Omron CX-Programmer project NuovoProgetto (CX-Programmer 9.61)

# PLC NewPLC1: CJ2M CPU32
I/O table (CPU CJ2M-CPU32): rack 0 slot 11 CJ2M-EIP21

## Global symbols (name address type ; comment)
AnnoNecessario D700 INT  ; 1° Word di lavoro - Anno di produzione
AnnoNecessarioRicetta D300 INT
AutCmdNotturno W20.07 BOOL
AutCmdStop W20.06 BOOL
AutFlagConforme W20.08 BOOL
AutPoupupAcido W21.02 BOOL
AutPoupupBedina D6122 INT
AutPoupupScolaggio W21.00 BOOL
AutPoupupTBedina D6123 INT
AutPrepBedina W20.08 BOOL
AutPupupInvioBotte D1100.04 BOOL
AutRicettaENd W21.01 BOOL
AutStsScolaggioEnd 6.08 BOOL
0.04 BOOL  ; PER VIS DISPLAY
10.00 BOOL  ; SPIA DISPLAY
10.01 BOOL  ; SPIA DISPLAY
10.03 BOOL  ; SPIA DISPLAY
11.00 BOOL  ; mixA
11.01 BOOL  ; in da rete
11.02 BOOL  ; acqua fredda
11.03 BOOL  ; mixB
11.06 BOOL  ; reset prenotazio
15.00 BOOL  ; ELETTROV_GENERALE
15.01 BOOL  ; EV SCOLAGGIO
15.04 BOOL  ; LUCE VERDE
15.05 BOOL  ; LUCE ROSSA
15.06 BOOL  ; elettrov. mix A
15.07 BOOL  ; ELETTROVALVOLA VAPORE
15.08 BOOL  ; EV SCARICO VASCA
15.09 BOOL  ; EV CARICO VASCA
15.10 BOOL  ; MARCIA AV
15.11 BOOL  ; RELE AGITATORE
15.12 BOOL  ; freno botte
15.13 BOOL  ; AUX POMPA
15.14 BOOL  ; AUX ROTAZ. FILTRO
15.15 BOOL  ; MARCIA IN
204.00 BOOL  ; PER_VIS_DISPLAY
207.00 BOOL  ; SPIA DISPLAY
207.01 BOOL  ; SPIA DISPLAY
20.09 BOOL  ; Fp carica
20.10 BOOL  ; Fp salva
20.11 BOOL  ; Fp start
20.12 BOOL  ; Fp pausa
211 CHANNEL  ; out per rete
212 CHANNEL  ; out per rete
213 CHANNEL  ; out per rete
220.00 BOOL  ; out per rete
220.01 BOOL  ; out per rete
220.02 BOOL  ; out per rete
220.03 BOOL  ; out per rete
220.04 BOOL  ; out per rete
220.05 BOOL  ; mixA
220.06 BOOL  ; mixB
28.01 BOOL  ; prenota
28.06 BOOL  ; check prenot acq
28.09 BOOL  ; conferma dati fo
28.10 BOOL  ; conferma dati gl
28.11 BOOL  ; tasto start form
28.12 BOOL  ; tasto stop formi
28.13 BOOL  ; tasto start glut
28.14 BOOL  ; tasto stop gluta
30.07 BOOL  ; SEGN. DISPLAY
38.04 BOOL  ; manuale filtro
38.05 BOOL  ; manuale mix B
38.07 BOOL  ; riciclo in attes
3.08 BOOL  ; Comando valvola vapore (?)
40.00 BOOL  ; attesa prenotazi
40.01 BOOL  ; acqua in macchin
40.02 BOOL  ; formico in uso
40.03 BOOL  ; solforico in uso
40.04 BOOL  ; glutaral in uso
40.05 BOOL  ; ingresso formico
40.06 BOOL  ; ingresso glutara
42 CHANNEL  ; Da DeviceNet: litri attuali erogati
6.14 BOOL  ; carico bagno
7.02 BOOL  ; tasto ACQUA
7.03 BOOL  ; a pg quantità
7.08 BOOL  ; on agitatore
7.09 BOOL  ; scarico bagno
8.10 BOOL  ; led formico
8.11 BOOL  ; led solforico
8.12 BOOL  ; led glutaral
9.00 BOOL  ; scelta formico
9.01 BOOL  ; scelta solforico
9.02 BOOL  ; scelta glutaral
9.15 BOOL  ; annullamento sce
D1210 CHANNEL  ; Setpoint litri in DEC
D1212 CHANNEL  ; Litri attuali in DEC
D1250 CHANNEL  ; Secondi mancanti
D1260 CHANNEL  ; Minuti per HMI
D214 CHANNEL  ; Puntatore step
D216 CHANNEL  ; Puntatore Step+1
D300 CHANNEL  ; Passo attuale
D3000 CHANNEL  ; Memoria H0
D3002 CHANNEL  ; Memoria D502
D3102 CHANNEL  ; Puntatore
D502 CHANNEL  ; Cambio pagina lato HMI
D58 CHANNEL  ; °C di erogazione
D59 CHANNEL  ; dec/lt in botte
D600 CHANNEL  ; Passo precedente
D700 CHANNEL  ; Passo successivo
D800 CHANNEL  ; Clear
D85 CHANNEL  ; set +
D86 CHANNEL  ; set -
D92 CHANNEL  ; numero botte
E21005 CHANNEL  ; Puntatore a passo da salvare
E21006 CHANNEL  ; Puntatore per caricamento passo da DB a lavoro
E22002 CHANNEL  ; Passo meno 1
H0 CHANNEL  ; Cambio pagina PLC
H12.00 BOOL  ; timer rotazione
H12.04 BOOL  ; sblocco di prova
H4.13 BOOL  ; relè carico bagn
H4.14 BOOL  ; relè agitatore
H4.15 BOOL  ; relè scarico bag
H5.11 BOOL  ; scarico esterno
H6.01 BOOL  ; start miscelazio
H6.02 BOOL  ; segn acqua in ri
H6.03 BOOL  ; segn acquaA in b
H6.05 BOOL  ; abbandono erogaz
H6.07 BOOL  ; segnalazione pre
H6.08 BOOL  ; start miscelazio
H6.09 BOOL  ; segn acquaB in b
T0140 BOOL  ; Delay discrepanza pagine
T0150 BOOL  ; Delay simulazione cmd acqua
T0151 BOOL  ; Delay simulazione cmd acido formico
T0152 BOOL  ; Delay reset feedback acido formico
T0153 BOOL  ; Delay simulazione cmd glutaraldeide
T0154 BOOL  ; Delay reset feedback glutaraldeide
T0156 BOOL  ; Simulazione riempimento acqua in corso
W24.02 BOOL  ; Memoria comando acqua
BedinaRunning D1103.00 BOOL  ; Preparazione bedina in corso
BedinaTimeEnd D1103.01 BOOL
BedinaTimeRef D1103.03 BOOL
BedinaTimeRun D1103.02 BOOL
CaricaRIcetta W20.01 BOOL  ; Carica ricetta
CmdAcqua 28.01 BOOL
CmdFormico 28.09 BOOL
CmdGlutaral 28.10 BOOL
CmdPIDon 2.11 BOOL
CmdRotAlt 3.01 BOOL
CmdRotAv 1.04 BOOL
CmdRotInd 1.05 BOOL
CmdRotNotte 3.13 BOOL
CmdRotStop 1.03 BOOL
CmdScolaggioDecrementoAsse 4.09 BOOL
CmdScolaggioNormale 4.08 BOOL
CmdTemperaturaOFF 2.13 BOOL
CmdTemperaturaON 2.12 BOOL
CodiceNecessario D750 DINT
CodiceNecessarioRicetta D350 DINT
ConfermaBarcodeLetto D1101.03 BOOL
ConfermaBedina D1100.00 BOOL
ConfermaControllo D1100.07 BOOL
ConfermaInvioBotte D1100.01 BOOL
ConfermaMancatoScolaggio D2000.09 BOOL
ConfermaRotNotte 3.15 BOOL
DelayRotazione D1000 UINT
FeedbackAcqua H6.03 BOOL
FeedbackFormico 40.05 BOOL
FeedbackGlutaral 40.06 BOOL
FeedbackRichiestaFormico 8.10 BOOL
FeedbackRotAlt H4.06 BOOL
FeedbackRotAv 207.00 BOOL
FeedbackRotInd 207.01 BOOL
FeedbackRotNotte 4.03 BOOL
FlagAbilitaScansioni D1810.04 BOOL
FlagIgnoraScansioniFallite D1810.02 BOOL
FlagNascondiTasti 1810.04 BOOL
FlagNuovaScansione D1810.00 BOOL
FlagPrimaScansione D1802.00 BOOL
FlagRiempimentoAcqua D2000.07 BOOL  ; =1 a fine riempimento acqua
FlagRitentaScansioni D1810.03 BOOL
FlagScansioniFallite D1810.01 BOOL
FlagSolido D1102.03 BOOL  ; Per fermata botte inserimento prodotti solidi
FlagStsEnd D1100.02 BOOL
GlobalGreenFlash D1102.02 BOOL
GlobalGreenLight D1102.01 BOOL
GlobalStsRun D1102.00 BOOL  ; =1 se ricetta AUT in marcia
LetturaBarcodeErrata D1101.01 BOOL
LetturaBarcodeOK D1101.02 BOOL
LetturaCodPro D1150 DINT  ; Codice letto da barcode
LetturaPesoDINT D1154 DINT  ; Peso letto da barcode (in INTERO)
LetturaPesoMem D1156 REAL
LetturaPesoREAL D1160 REAL  ; Peso letto da barcode (in REALE)
LetturaRicetta D1152 DINT
LetturaRicettaTemp D1162 DINT
LitriAcqua D57 WORD
MemCodPro D1802 DINT
MemPeso D1806 REAL
MemRicetta D1804 DINT
MemTimSkip D2000.05 BOOL
MinAltPreNotte D40 INT  ; Minuti prima di attivare alternata notte
NumeroScansioni D1808 INT
OreAltPreNotte D39 INT  ; Ore prima di attivare alternata notte
PaginaAtt D502 INT
PassoPuntatore D3100 CHANNEL  ; Passo
PassoPuntatoreINT D3106 INT
PercentualeREAL D1164 REAL
PesoFormico D82 WORD
PesoGlutaral D83 WORD
PesoNecessario D760 REAL
PesoNecessarioRicetta D360 REAL
PopupMancatoScolaggio D2000.08 BOOL  ; =1 se viene attivato un riempimento acqua  e FlagRiempimentoAcqua è già TRUE
PopupRotNotte D2000.04 BOOL
ProdottoErratoIgnora D1101.06 BOOL
ProdottoErratoPopup D1101.05 BOOL
ProdottoErratoRiprova 1101.07 BOOL
PupConfermaInvioBotte D1100.03 BOOL
REAL1000 D1166 REAL
RicAaSca D8000 WORD  ; 1° Word di lavoro - Anno di produzione
RicAzione D8006 WORD  ; Codice azione
RicBotte D8003 WORD  ; Bottale (1-10) di destinazione
RicCheck D8074 WORD  ; Tipo controllo: 1=PH 2=Colore 3=Penetrazione
RicCodPro D8050 DWORD  ; Codice prodotto
RicDescr D8007 STRING[40]  ; Descrizione azione
RicGradi D8064 WORD  ; Temperatura acqua
RicLoaded D8092.00 BOOL  ; 0=nuova 1=ricetta importata
RicMax D8080 REAL  ; Valore massimo per controllo
RicMin D8076 REAL  ; Valore minimo per controllo
RicMinuti D8066 WORD  ; Minuti di rotazione
RicNumSca D8001 DWORD  ; Progressivo ricetta
RicPause W20.04 BOOL  ; Pausa ricetta
RicPeso D8060 REAL  ; Peso prodotto in Kg
RicRata D8054 WORD  ; 1=Raggruppamento prodotti
RicRigNum D8004 WORD  ; Numero progressivo riga
RicRigSot D8005 WORD  ; Numero progressivo sottoriga
RicRilevato D8084 REAL  ; Valore rilevato al controllo
RicRotaz D8068 WORD  ; Tipo di rotazione
RicScola D8070 WORD  ; Tipo di scolatura
RicSpeed D8072 WORD  ; Velocità (da 2 a 8)
RicStart W20.03 BOOL  ; Start ricetta
RicStato D8088 WORD  ; Stato riga
RicStatus D510 WORD
RicStsRun W20.05 BOOL  ; RicStsRun
RicTipPro D8056 WORD  ; L/76=Liquido S/83=Solido
RicUser D8090 WORD  ; ID Utente che convalida la riga
RicValvola D8058 WORD  ; Valvola associata al prodotto
RicettaNecessaria D701 DINT  ; Progressivo ricetta
RicettaNecessariaRicetta D301 DINT
RichiestaConfermaBedina D1101.04 BOOL
RichiestaFormico 9.00 BOOL
RichiestaGlutar 28.08 BOOL
RichiestaLetturaBarcode D1101.00 BOOL
SalvaRicetta W20.00 BOOL  ; Salva ricetta
SceltaFormico 28.07 BOOL
SceltaGlutar 9.02 BOOL
SkipPasso W20.02 BOOL  ; Salta al passo successivo
StatoMacchina D4000 INT
StatoScansione D1800 INT
StsScolaggioDecrementoAsse 5.01 BOOL
StsScolaggioNormale 5.00 BOOL
TempReal D1008 REAL
TemperaturaAcqua D56 CHANNEL
TemperaturaAcquaPerBCD D3200 CHANNEL
TemperaturaMacchina D23 CHANNEL
TimerAcqua1 T0080 TIMER
TimerAcqua2 T0081 TIMER
TimerAcqua3 T0082 TIMER
TimerAcqua4 T0083 TIMER
TimerFormico1 T0070 TIMER
TimerFormico2 T0071 TIMER
TimerFormico3 T0072 TIMER
TimerFormico4 T0073 TIMER
TimerFormico5 T0074 TIMER
TimerFormico6 T0075 TIMER
TimerGlutar1 T0084 TIMER
TimerGlutar2 T0085 TIMER
TimerGlutar3 T0086 TIMER
TimerGlutar4 T0087 TIMER
TimerGlutar5 T0088 TIMER
TimerGlutar6 T0089 TIMER
TimerPIDoff T0100 TIMER
TimerPIDon T0099 TIMER
TimerRotazione T0093 TIMER
TimerRotazione3 T0094 TIMER
TimerRotazione4 T0095 TIMER
TimerRotazione6 T0096 TIMER
TimerRotazione7 T0097 TIMER
TimerRotazione8 T0098 TIMER
TimerSaltaPasso T0102 TIMER  ; 1s minimo per salto passo
TimerScolaggioNormale T0105 TIMER
TimerScolaggioON T0101 TIMER
TimxBedinaDelay D1206 INT
TimxNumeroOre D1200 INT
TimxRicMinuti D1202 INT
TimxTempDelay D1201 INT
Tolleranza D1140 REAL
TolleranzaInf D1144 REAL
TolleranzaSup D1142 REAL
VaiAInvioInBotte D1100.06 BOOL
VelocBotte D1004 WORD
VisibilitàIndietroMan D2000.06 BOOL  ; Visualizza o meno la freccia indietro verso manuale in HMI
acqua_litriErogati D1212 INT
acqua_setpointRicetta D1210 INT
annullaRicetta D1810.11 BOOL
barrieraAperta W24.08 BOOL
barrieraChiusa W24.09 BOOL
barrieraDigIn 14.03 BOOL
cmdScolaggioBotte W24.05 BOOL  ; Comando per scolaggio da procedura solo botte
confermaVaiABedina D1810.08 BOOL
delayAlternataOn W20.14 BOOL
delayPopupControllo T0106 TIMER
flagFineScolaggio D1810.07 BOOL
flagPrimoRiempimento D1810.14 BOOL  ; =1 dopo il primo riempimento d'acqua. torna a 0 dopo uno scolaggio
inserimentoProdottiRunning D1180.09 BOOL
instCreaData creaData
invioConRisciacquoON H4.15 BOOL
invioSenzaRisciacquoON H5.08 BOOL
luceProdotti D100.00 BOOL
memCmdFormico W24.00 BOOL  ; Memoria cmd formico
memCmdGlutaraldeide W24.01 BOOL  ; Memoria cmd glutaraldeide
minutiRimanentiAlternata D31 CHANNEL
offsetRiga1 D1830 INT
offsetRiga2 D1831 INT
offsetRiga3 D1832 INT
offsetRiga4 D1833 INT
offsetRiga5 D1834 INT
offsetRiga6 D1835 INT
popupConfScola W24.07 BOOL
popupPresOpScola W24.06 BOOL
presenzaOpAcido D1810.06 BOOL  ; Conferma presenza operatore per invio acido/glutaral.
rRicStsRun H50.00 BOOL
scrollDown D1810.10 BOOL
scrollUp D1810.09 BOOL
secondiRimanentiAlternata D30 CHANNEL
stopDaBarriera 6.03 BOOL
tempCondStep1 W20.12 BOOL
temperaturaAcquaErogata 43 WORD
temperaturaBotte 2005 WORD
tempoChiamataOperatore D1820 INT
tempoPasso D1836 INT
tempoPassoMem D1837 INT
timerAlternata T0190 TIMER
timerScrollDown T0108 TIMER
timerScrollUp T0107 TIMER
visibPopupPulsanti D1103.04 BOOL  ; Visibilità pulsanti di conferma su pagina automatico
visualizzaKgAcido W24.03 BOOL
visualizzaKgGlutaral W24.04 BOOL

## Program NuovoProgramma1 (cyclic task 0)
Local symbols
BARRIERA_SIC 14.03 BOOL
EMERGENZA_ARIA 14.00 BOOL
LIVELLO_VASCA 14.04 BOOL
PROX_POS 14.01 BOOL
TERMICI 14.02 BOOL

### Section Sezione1

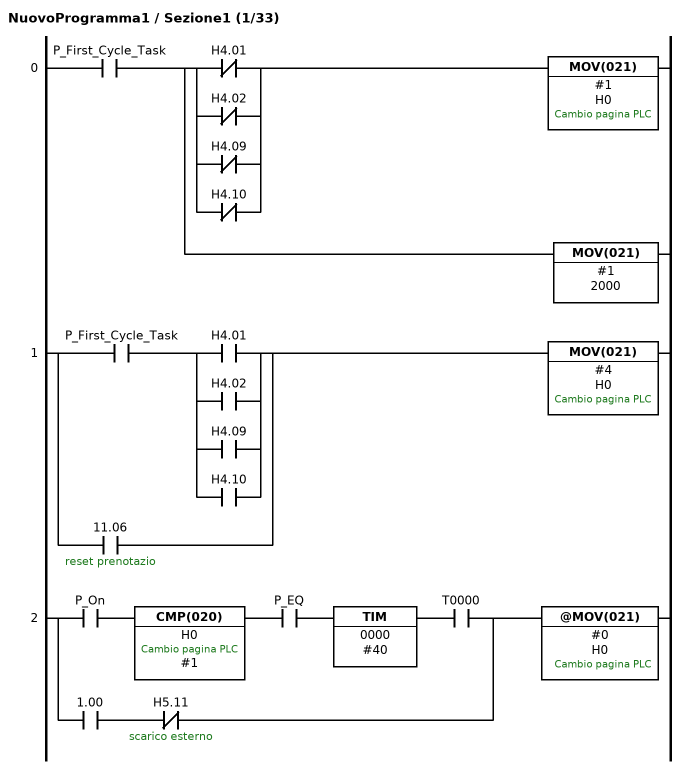
; rung 0
LD P_First_Cycle_Task
OUT TR0
LDNOT H4.01
ORNOT H4.02
ORNOT H4.09
ORNOT H4.10
ANDLD
MOV(021) #1 H0  ; Cambio pagina PLC
LD TR0
MOV(021) #1 2000
; rung 1
LD P_First_Cycle_Task
LD H4.01
OR H4.02
OR H4.09
OR H4.10
ANDLD
OR 11.06  ; reset prenotazio
MOV(021) #4 H0  ; Cambio pagina PLC
; rung 2
LD P_On
CMP(020) H0 #1  ; Cambio pagina PLC
AND P_EQ
TIM 0000 #40
AND T0000
LD 1.00
ANDNOT H5.11  ; scarico esterno
ORLD
@MOV(021) #0 H0  ; Cambio pagina PLC

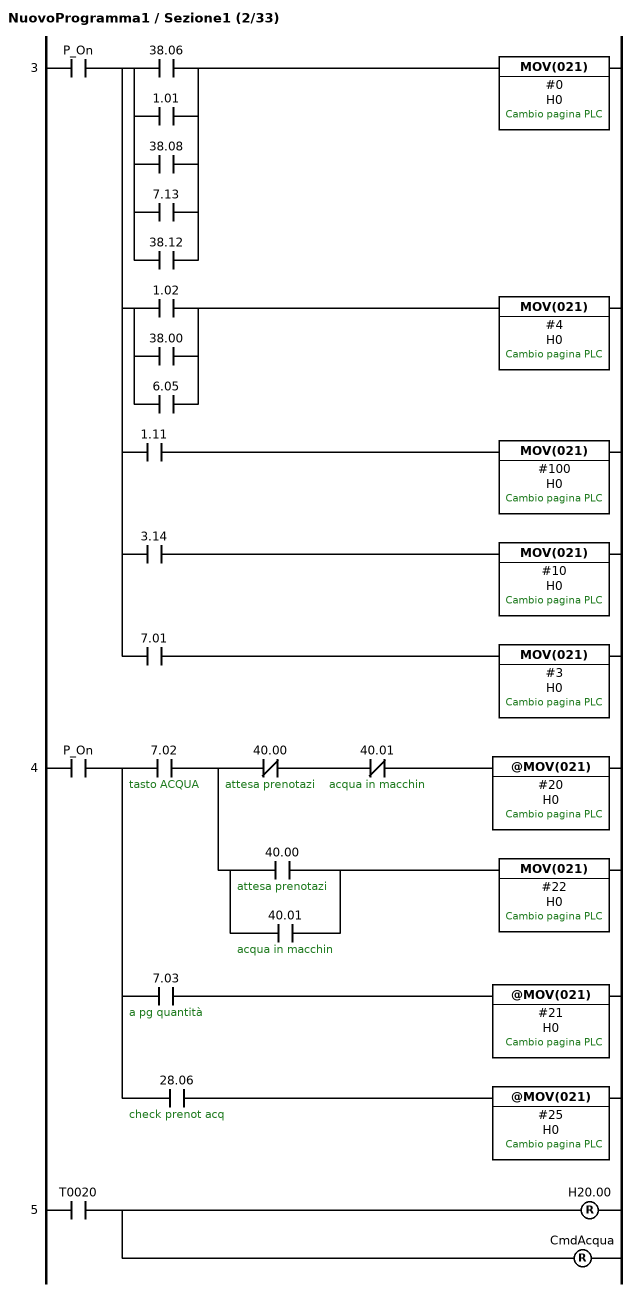
; rung 3
LD P_On
OUT TR0
LD 38.06
OR 1.01
OR 38.08
OR 7.13
OR 38.12
ANDLD
MOV(021) #0 H0  ; Cambio pagina PLC
LD TR0
LD 1.02
OR 38.00
OR 6.05
ANDLD
MOV(021) #4 H0  ; Cambio pagina PLC
LD TR0
AND 1.11
MOV(021) #100 H0  ; Cambio pagina PLC
LD TR0
AND 3.14
MOV(021) #10 H0  ; Cambio pagina PLC
LD TR0
AND 7.01
MOV(021) #3 H0  ; Cambio pagina PLC
; rung 4
LD P_On
OUT TR0
AND 7.02  ; tasto ACQUA
OUT TR1
ANDNOT 40.00  ; attesa prenotazi
ANDNOT 40.01  ; acqua in macchin
@MOV(021) #20 H0  ; Cambio pagina PLC
LD TR1
LD 40.00  ; attesa prenotazi
OR 40.01  ; acqua in macchin
ANDLD
MOV(021) #22 H0  ; Cambio pagina PLC
LD TR0
AND 7.03  ; a pg quantità
@MOV(021) #21 H0  ; Cambio pagina PLC
LD TR0
AND 28.06  ; check prenot acq
@MOV(021) #25 H0  ; Cambio pagina PLC
; rung 5
LD T0020
RSET H20.00
RSET CmdAcqua

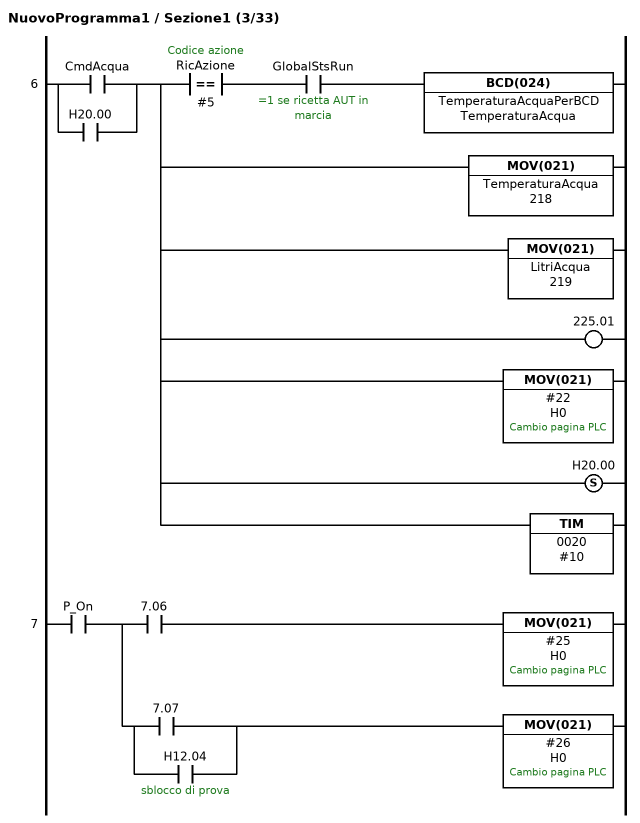
; rung 6
LD CmdAcqua
OR H20.00
OUT TR0
AND=(300) RicAzione #5  ; Codice azione
AND GlobalStsRun  ; =1 se ricetta AUT in marcia
BCD(024) TemperaturaAcquaPerBCD TemperaturaAcqua
LD TR0
MOV(021) TemperaturaAcqua 218
MOV(021) LitriAcqua 219
OUT 225.01
MOV(021) #22 H0  ; Cambio pagina PLC
SET H20.00
TIM 0020 #10
; rung 7
LD P_On
OUT TR0
AND 7.06
MOV(021) #25 H0  ; Cambio pagina PLC
LD TR0
LD 7.07
OR H12.04  ; sblocco di prova
ANDLD
MOV(021) #26 H0  ; Cambio pagina PLC

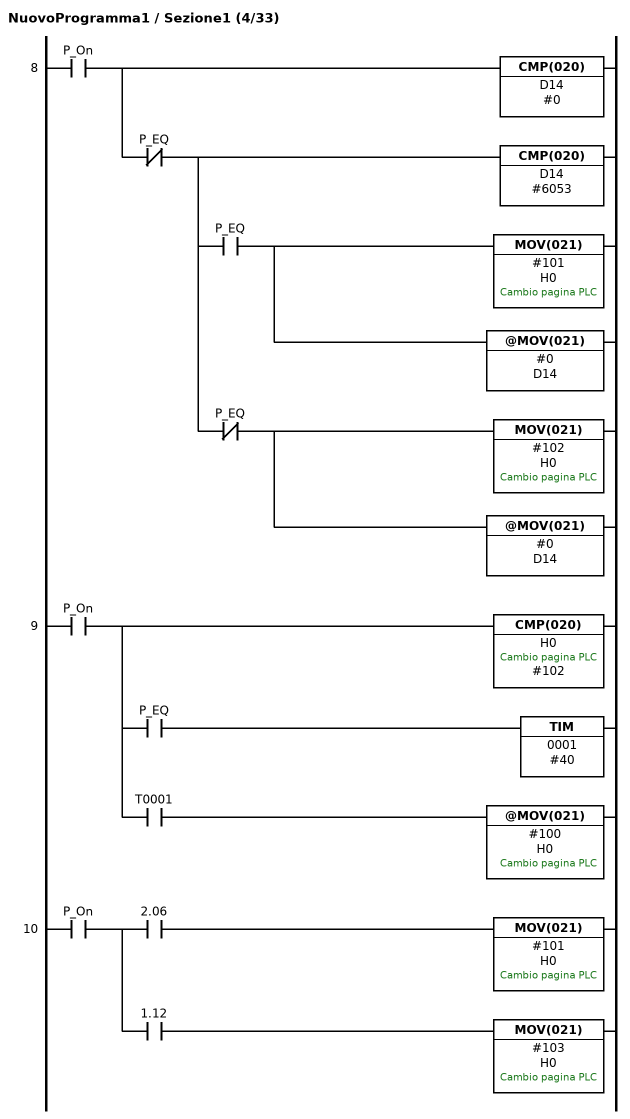
; rung 8
LD P_On
CMP(020) D14 #0
ANDNOT P_EQ
OUT TR0
CMP(020) D14 #6053
AND P_EQ
MOV(021) #101 H0  ; Cambio pagina PLC
@MOV(021) #0 D14
LD TR0
ANDNOT P_EQ
MOV(021) #102 H0  ; Cambio pagina PLC
@MOV(021) #0 D14
; rung 9
LD P_On
OUT TR0
CMP(020) H0 #102  ; Cambio pagina PLC
AND P_EQ
TIM 0001 #40
LD TR0
AND T0001
@MOV(021) #100 H0  ; Cambio pagina PLC
; rung 10
LD P_On
OUT TR0
AND 2.06
MOV(021) #101 H0  ; Cambio pagina PLC
LD TR0
AND 1.12
MOV(021) #103 H0  ; Cambio pagina PLC

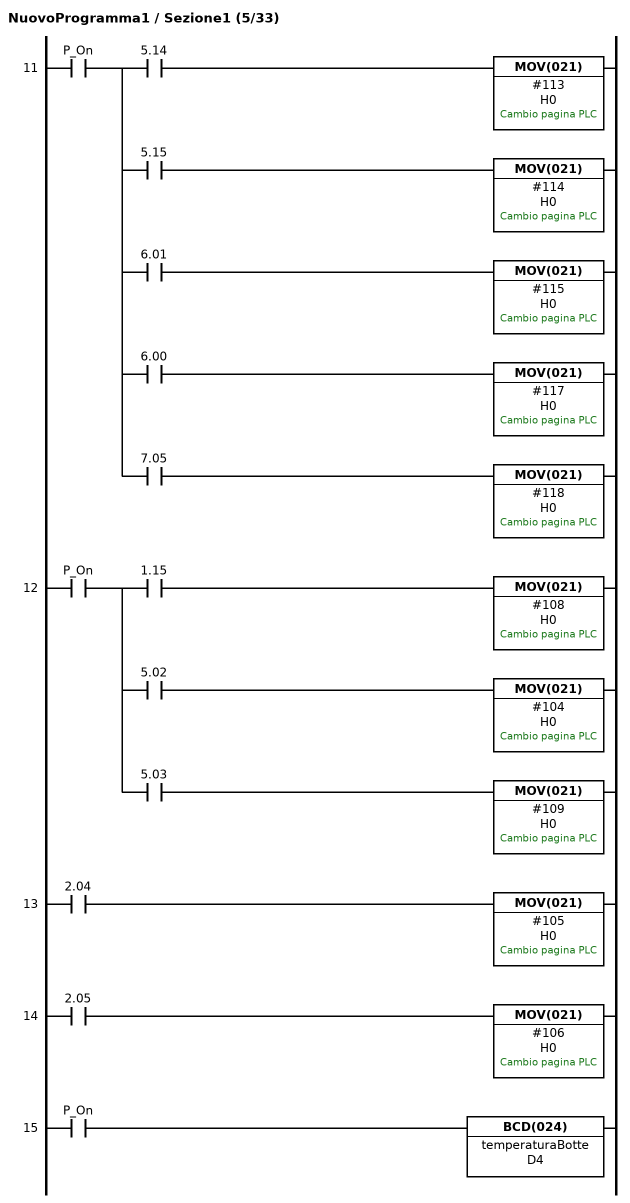
; rung 11
LD P_On
OUT TR0
AND 5.14
MOV(021) #113 H0  ; Cambio pagina PLC
LD TR0
AND 5.15
MOV(021) #114 H0  ; Cambio pagina PLC
LD TR0
AND 6.01
MOV(021) #115 H0  ; Cambio pagina PLC
LD TR0
AND 6.00
MOV(021) #117 H0  ; Cambio pagina PLC
LD TR0
AND 7.05
MOV(021) #118 H0  ; Cambio pagina PLC
; rung 12
LD P_On
OUT TR0
AND 1.15
MOV(021) #108 H0  ; Cambio pagina PLC
LD TR0
AND 5.02
MOV(021) #104 H0  ; Cambio pagina PLC
LD TR0
AND 5.03
MOV(021) #109 H0  ; Cambio pagina PLC
; rung 13
LD 2.04
MOV(021) #105 H0  ; Cambio pagina PLC
; rung 14
LD 2.05
MOV(021) #106 H0  ; Cambio pagina PLC
; rung 15
LD P_On
BCD(024) temperaturaBotte D4

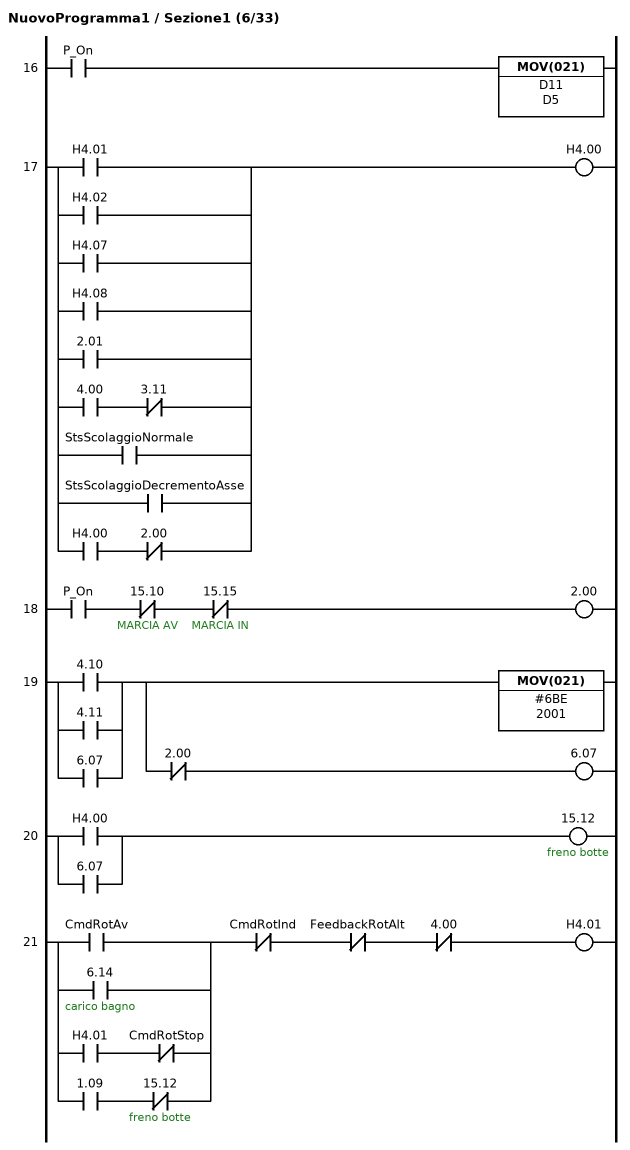
; rung 16
LD P_On
MOV(021) D11 D5
; rung 17
LD H4.01
OR H4.02
OR H4.07
OR H4.08
OR 2.01
LD 4.00
ANDNOT 3.11
ORLD
OR StsScolaggioNormale
OR StsScolaggioDecrementoAsse
LD H4.00
ANDNOT 2.00
ORLD
OUT H4.00
; rung 18
LD P_On
ANDNOT 15.10  ; MARCIA AV
ANDNOT 15.15  ; MARCIA IN
OUT 2.00
; rung 19
LD 4.10
OR 4.11
OR 6.07
MOV(021) #6BE 2001
ANDNOT 2.00
OUT 6.07
; rung 20
LD H4.00
OR 6.07
OUT 15.12  ; freno botte
; rung 21
LD CmdRotAv
OR 6.14  ; carico bagno
LD H4.01
ANDNOT CmdRotStop
ORLD
LD 1.09
ANDNOT 15.12  ; freno botte
ORLD
ANDNOT CmdRotInd
ANDNOT FeedbackRotAlt
ANDNOT 4.00
OUT H4.01

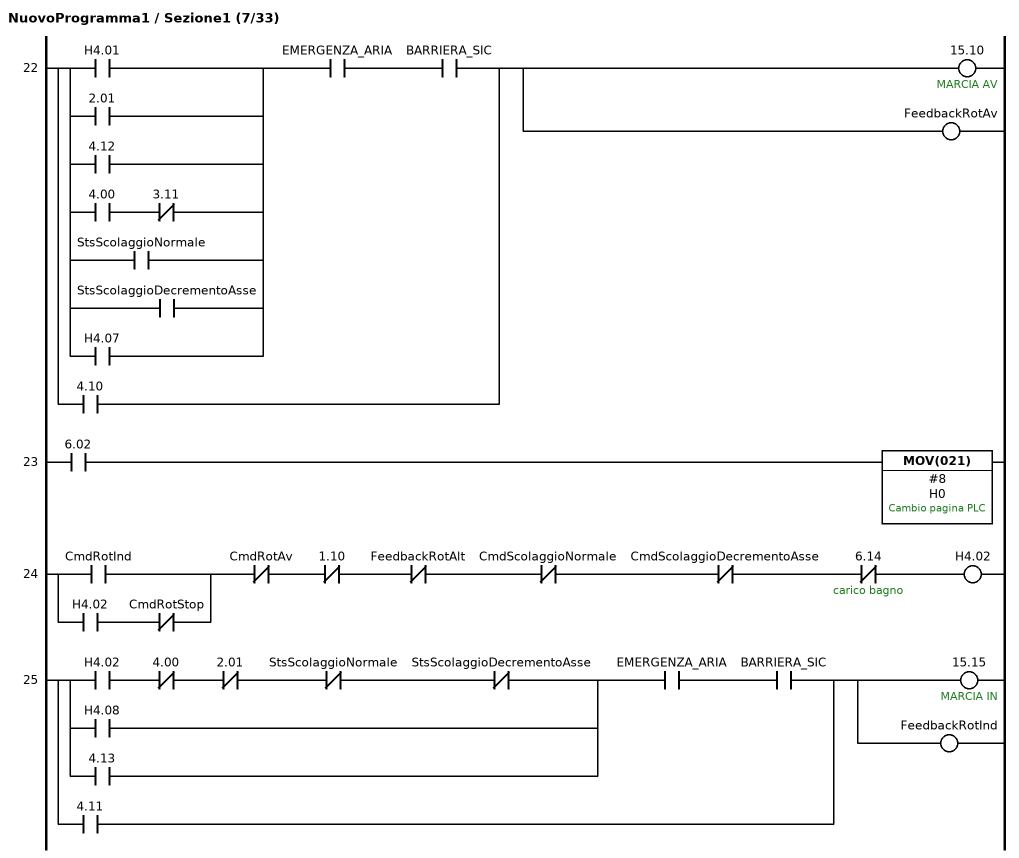
; rung 22
LD H4.01
OR 2.01
OR 4.12
LD 4.00
ANDNOT 3.11
ORLD
OR StsScolaggioNormale
OR StsScolaggioDecrementoAsse
OR H4.07
AND EMERGENZA_ARIA
AND BARRIERA_SIC
OR 4.10
OUT 15.10  ; MARCIA AV
OUT FeedbackRotAv
; rung 23
LD 6.02
MOV(021) #8 H0  ; Cambio pagina PLC
; rung 24
LD CmdRotInd
LD H4.02
ANDNOT CmdRotStop
ORLD
ANDNOT CmdRotAv
ANDNOT 1.10
ANDNOT FeedbackRotAlt
ANDNOT CmdScolaggioNormale
ANDNOT CmdScolaggioDecrementoAsse
ANDNOT 6.14  ; carico bagno
OUT H4.02
; rung 25
LD H4.02
ANDNOT 4.00
ANDNOT 2.01
ANDNOT StsScolaggioNormale
ANDNOT StsScolaggioDecrementoAsse
OR H4.08
OR 4.13
AND EMERGENZA_ARIA
AND BARRIERA_SIC
OR 4.11
OUT 15.15  ; MARCIA IN
OUT FeedbackRotInd

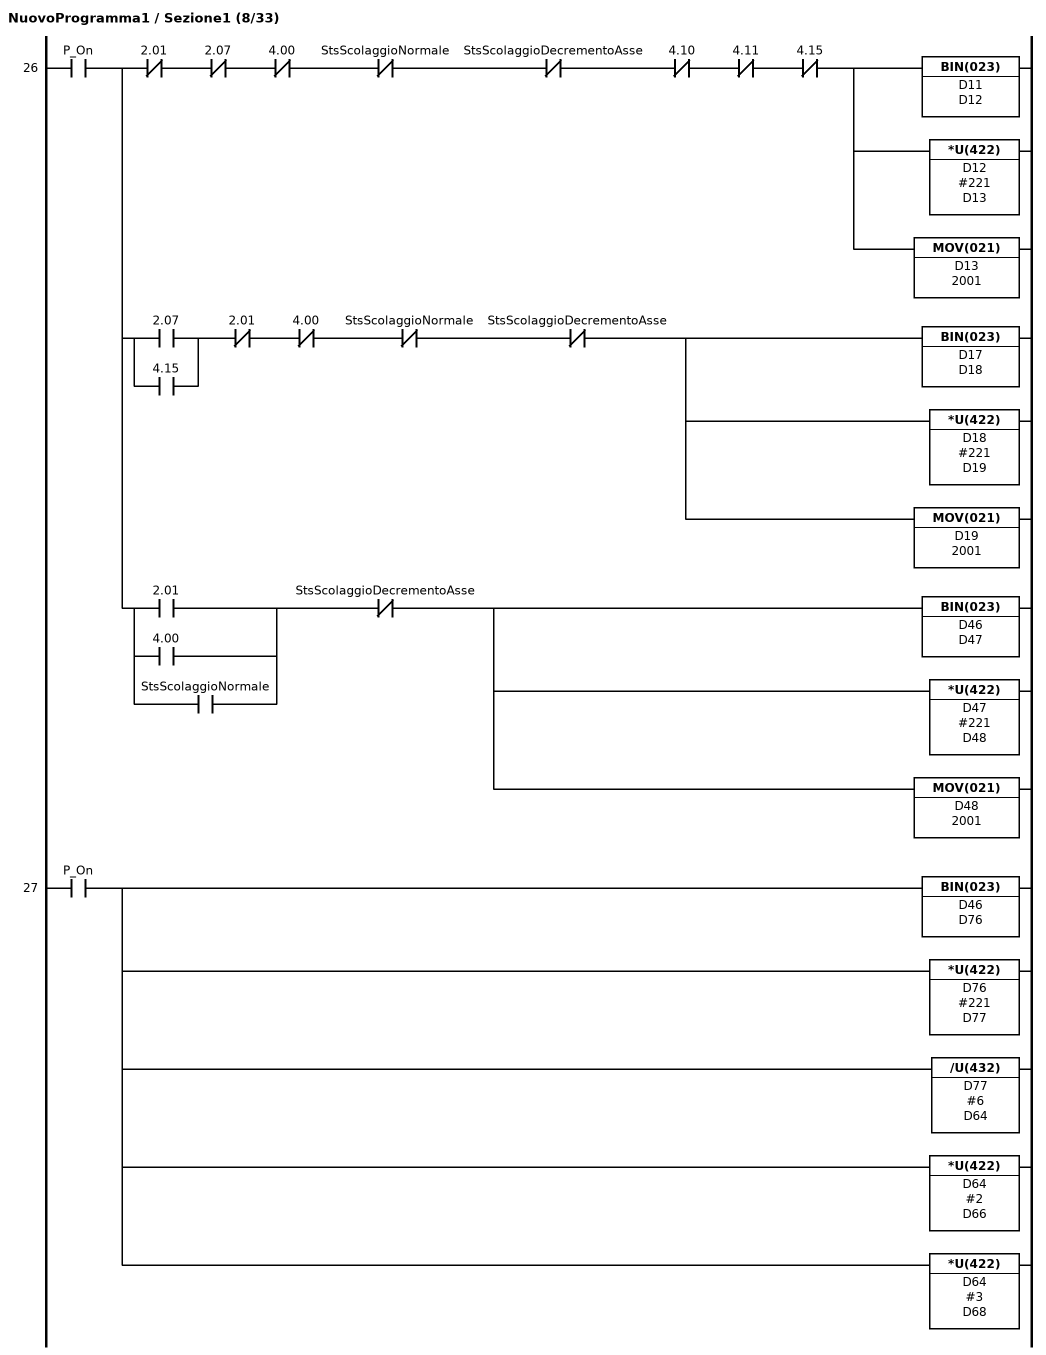
; rung 26
LD P_On
OUT TR0
ANDNOT 2.01
ANDNOT 2.07
ANDNOT 4.00
ANDNOT StsScolaggioNormale
ANDNOT StsScolaggioDecrementoAsse
ANDNOT 4.10
ANDNOT 4.11
ANDNOT 4.15
BIN(023) D11 D12
*U(422) D12 #221 D13
MOV(021) D13 2001
LD TR0
LD 2.07
OR 4.15
ANDLD
ANDNOT 2.01
ANDNOT 4.00
ANDNOT StsScolaggioNormale
ANDNOT StsScolaggioDecrementoAsse
BIN(023) D17 D18
*U(422) D18 #221 D19
MOV(021) D19 2001
LD TR0
LD 2.01
OR 4.00
OR StsScolaggioNormale
ANDLD
ANDNOT StsScolaggioDecrementoAsse
BIN(023) D46 D47
*U(422) D47 #221 D48
MOV(021) D48 2001
; rung 27
LD P_On
BIN(023) D46 D76
*U(422) D76 #221 D77
/U(432) D77 #6 D64
*U(422) D64 #2 D66
*U(422) D64 #3 D68

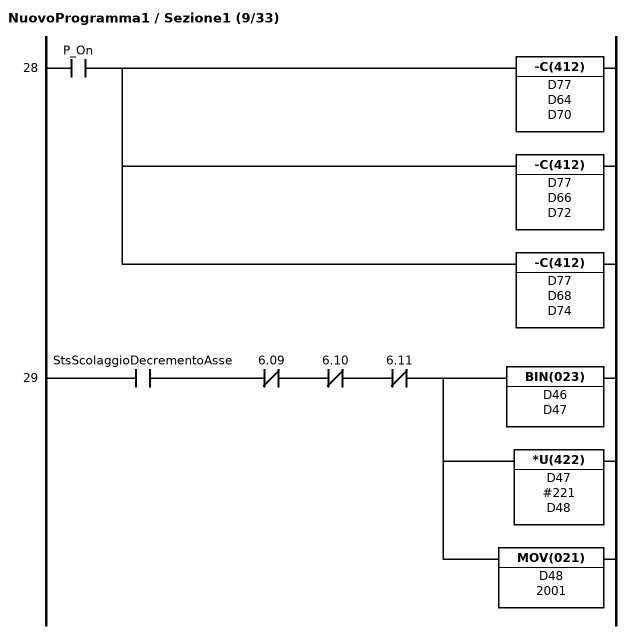
; rung 28
LD P_On
-C(412) D77 D64 D70
-C(412) D77 D66 D72
-C(412) D77 D68 D74
; rung 29
LD StsScolaggioDecrementoAsse
ANDNOT 6.09
ANDNOT 6.10
ANDNOT 6.11
BIN(023) D46 D47
*U(422) D47 #221 D48
MOV(021) D48 2001

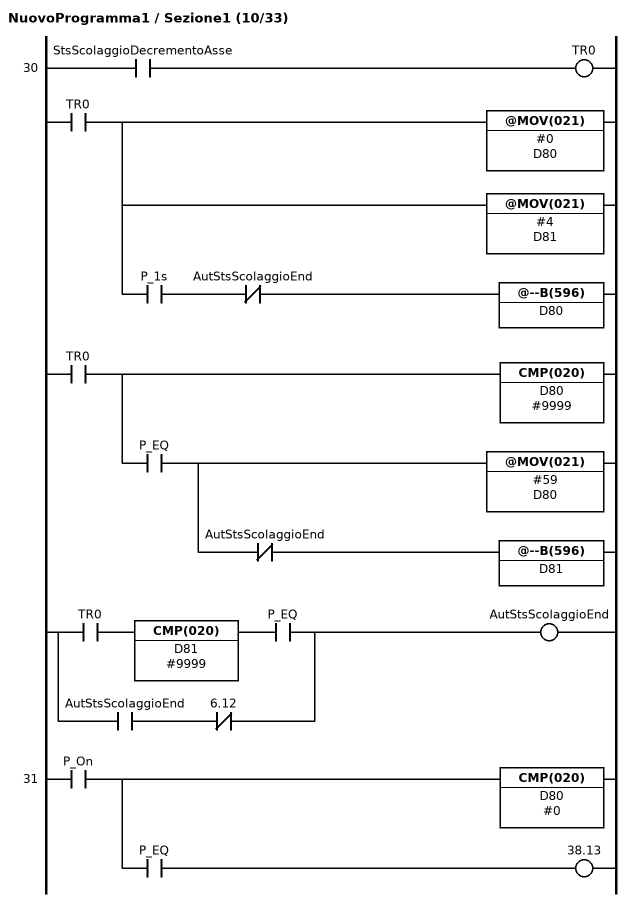
; rung 30
LD StsScolaggioDecrementoAsse
OUT TR0
@MOV(021) #0 D80
@MOV(021) #4 D81
AND P_1s
ANDNOT AutStsScolaggioEnd
@--B(596) D80
LD TR0
CMP(020) D80 #9999
AND P_EQ
@MOV(021) #59 D80
ANDNOT AutStsScolaggioEnd
@--B(596) D81
LD TR0
CMP(020) D81 #9999
AND P_EQ
LD AutStsScolaggioEnd
ANDNOT 6.12
ORLD
OUT AutStsScolaggioEnd
; rung 31
LD P_On
CMP(020) D80 #0
AND P_EQ
OUT 38.13

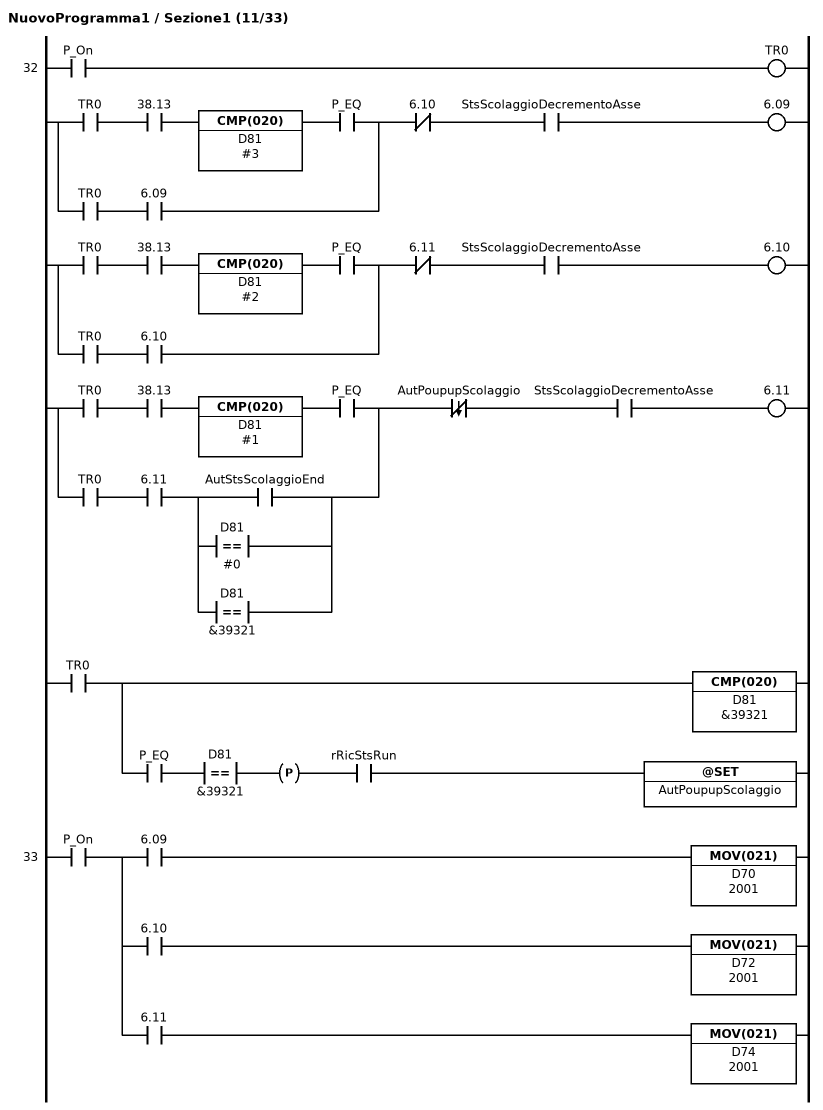
; rung 32
LD P_On
OUT TR0
AND 38.13
CMP(020) D81 #3
AND P_EQ
LD TR0
AND 6.09
ORLD
ANDNOT 6.10
AND StsScolaggioDecrementoAsse
OUT 6.09
LD TR0
AND 38.13
CMP(020) D81 #2
AND P_EQ
LD TR0
AND 6.10
ORLD
ANDNOT 6.11
AND StsScolaggioDecrementoAsse
OUT 6.10
LD TR0
AND 38.13
CMP(020) D81 #1
AND P_EQ
LD TR0
AND 6.11
LD AutStsScolaggioEnd
OR=(300) D81 #0
OR=(300) D81 &39321
ANDLD
ORLD
%ANDNOT AutPoupupScolaggio
AND StsScolaggioDecrementoAsse
OUT 6.11
LD TR0
CMP(020) D81 &39321
AND P_EQ
AND=(300) D81 &39321
UP(521)
AND rRicStsRun
@SET AutPoupupScolaggio
; rung 33
LD P_On
OUT TR0
AND 6.09
MOV(021) D70 2001
LD TR0
AND 6.10
MOV(021) D72 2001
LD TR0
AND 6.11
MOV(021) D74 2001

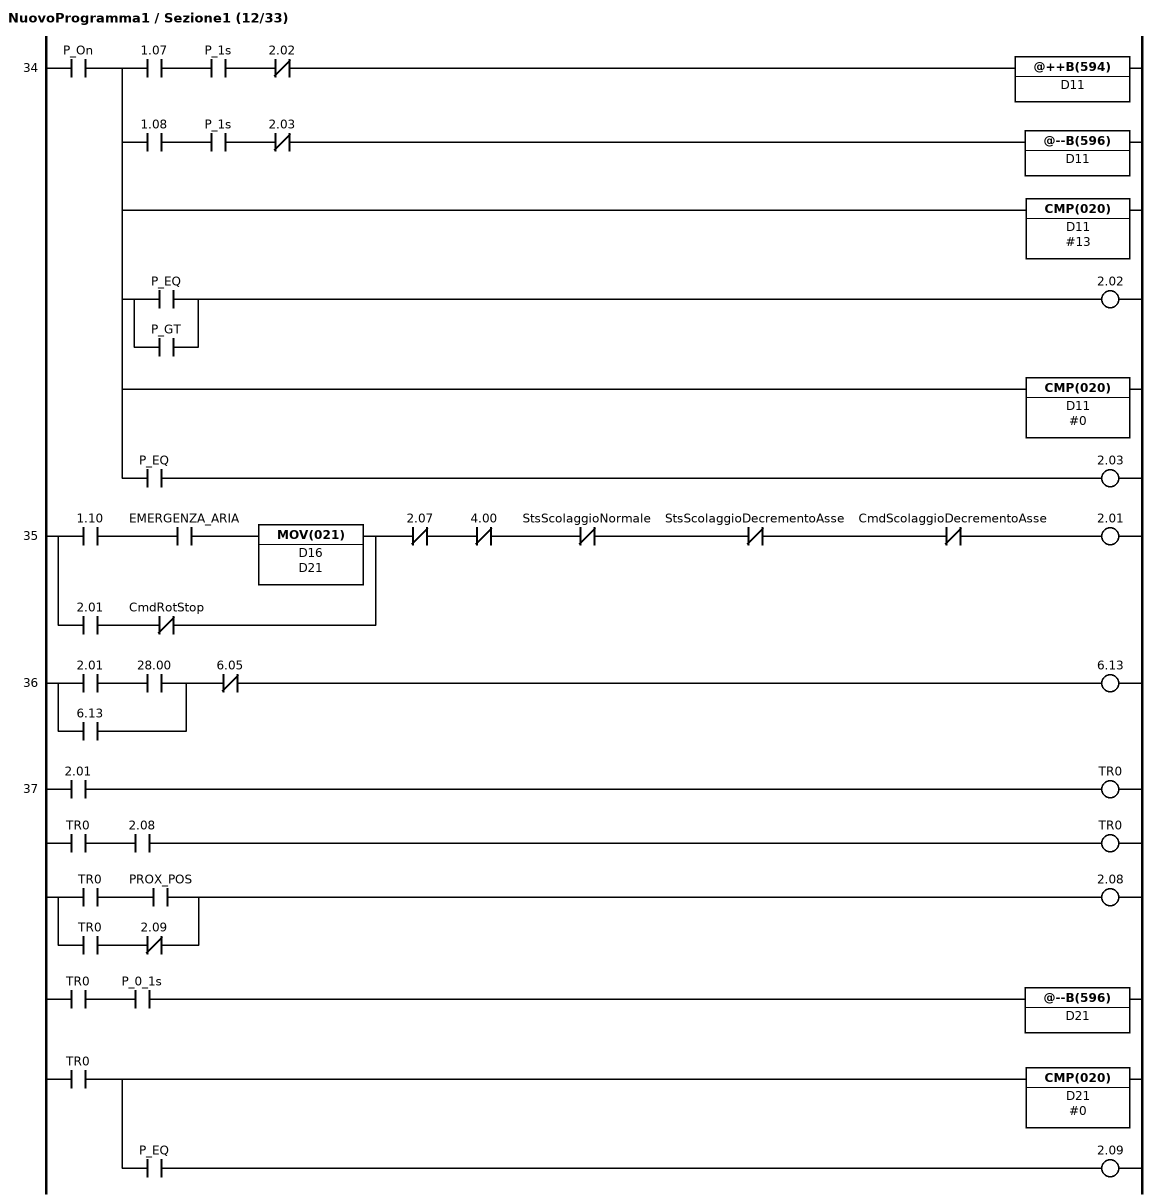
; rung 34
LD P_On
OUT TR0
AND 1.07
AND P_1s
ANDNOT 2.02
@++B(594) D11
LD TR0
AND 1.08
AND P_1s
ANDNOT 2.03
@--B(596) D11
LD TR0
CMP(020) D11 #13
LD P_EQ
OR P_GT
ANDLD
OUT 2.02
LD TR0
CMP(020) D11 #0
AND P_EQ
OUT 2.03
; rung 35
LD 1.10
AND EMERGENZA_ARIA
MOV(021) D16 D21
LD 2.01
ANDNOT CmdRotStop
ORLD
ANDNOT 2.07
ANDNOT 4.00
ANDNOT StsScolaggioNormale
ANDNOT StsScolaggioDecrementoAsse
ANDNOT CmdScolaggioDecrementoAsse
OUT 2.01
; rung 36
LD 2.01
AND 28.00
OR 6.13
ANDNOT 6.05
OUT 6.13
; rung 37
LD 2.01
OUT TR0
AND PROX_POS
LD TR0
AND 2.08
OUT TR0
ANDNOT 2.09
ORLD
OUT 2.08
LD TR0
AND P_0_1s
@--B(596) D21
LD TR0
CMP(020) D21 #0
AND P_EQ
OUT 2.09

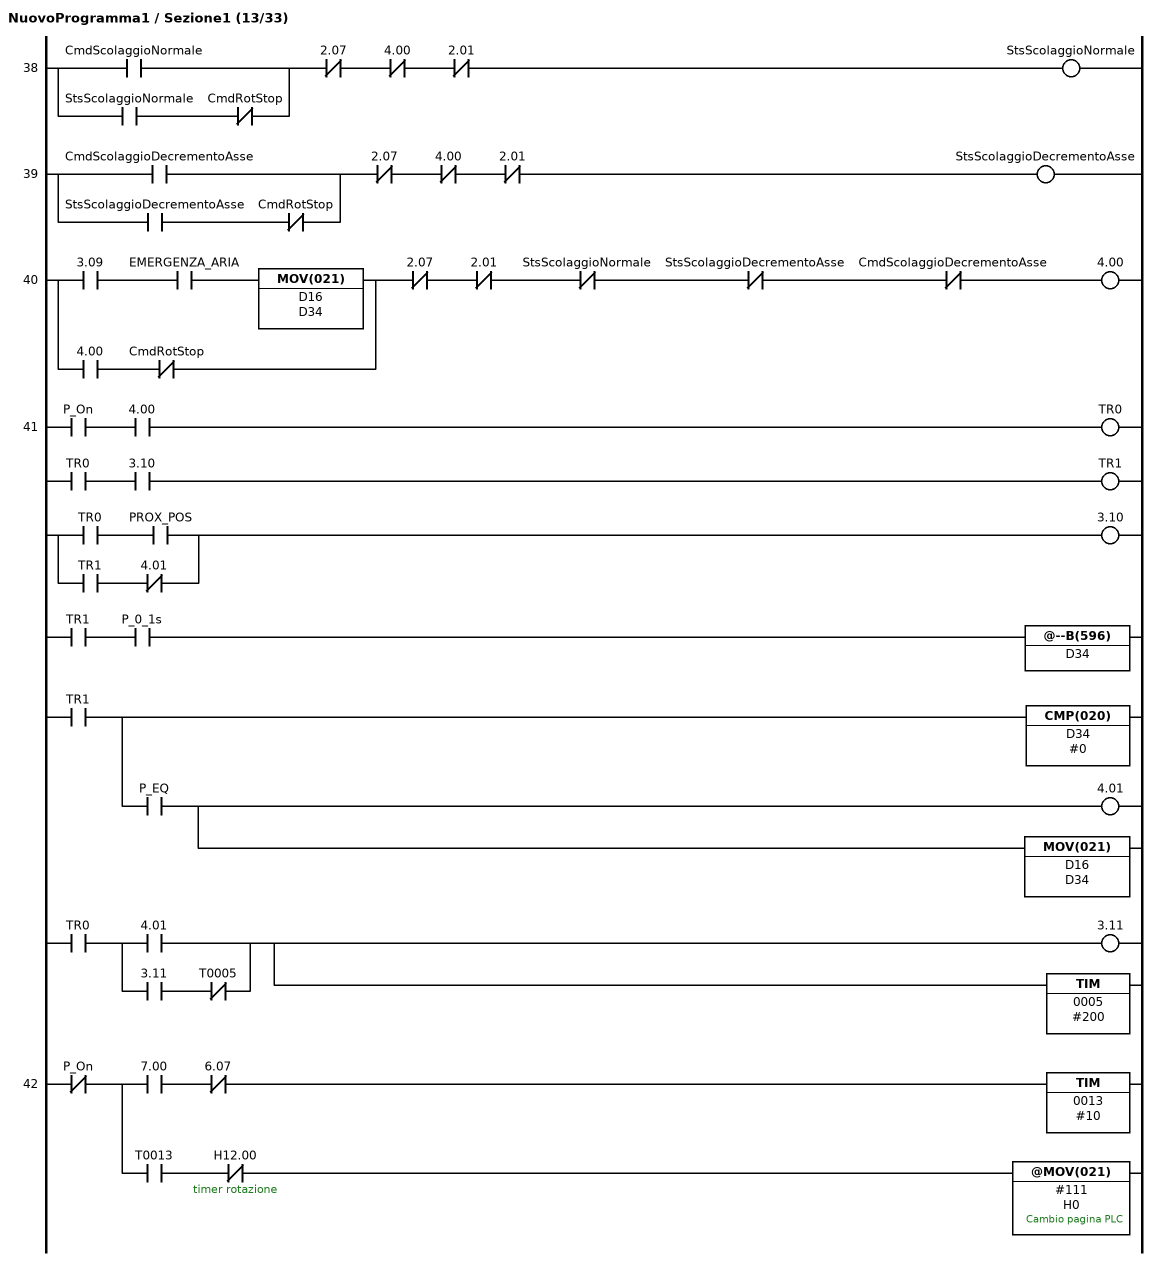
; rung 38
LD CmdScolaggioNormale
LD StsScolaggioNormale
ANDNOT CmdRotStop
ORLD
ANDNOT 2.07
ANDNOT 4.00
ANDNOT 2.01
OUT StsScolaggioNormale
; rung 39
LD CmdScolaggioDecrementoAsse
LD StsScolaggioDecrementoAsse
ANDNOT CmdRotStop
ORLD
ANDNOT 2.07
ANDNOT 4.00
ANDNOT 2.01
OUT StsScolaggioDecrementoAsse
; rung 40
LD 3.09
AND EMERGENZA_ARIA
MOV(021) D16 D34
LD 4.00
ANDNOT CmdRotStop
ORLD
ANDNOT 2.07
ANDNOT 2.01
ANDNOT StsScolaggioNormale
ANDNOT StsScolaggioDecrementoAsse
ANDNOT CmdScolaggioDecrementoAsse
OUT 4.00
; rung 41
LD P_On
AND 4.00
OUT TR0
AND PROX_POS
LD TR0
AND 3.10
OUT TR1
ANDNOT 4.01
ORLD
OUT 3.10
LD TR1
AND P_0_1s
@--B(596) D34
LD TR1
CMP(020) D34 #0
AND P_EQ
OUT 4.01
MOV(021) D16 D34
LD TR0
LD 4.01
LD 3.11
ANDNOT T0005
ORLD
ANDLD
OUT 3.11
TIM 0005 #200
; rung 42
LDNOT P_On
OUT TR0
AND 7.00
ANDNOT 6.07
TIM 0013 #10
LD TR0
AND T0013
ANDNOT H12.00  ; timer rotazione
@MOV(021) #111 H0  ; Cambio pagina PLC

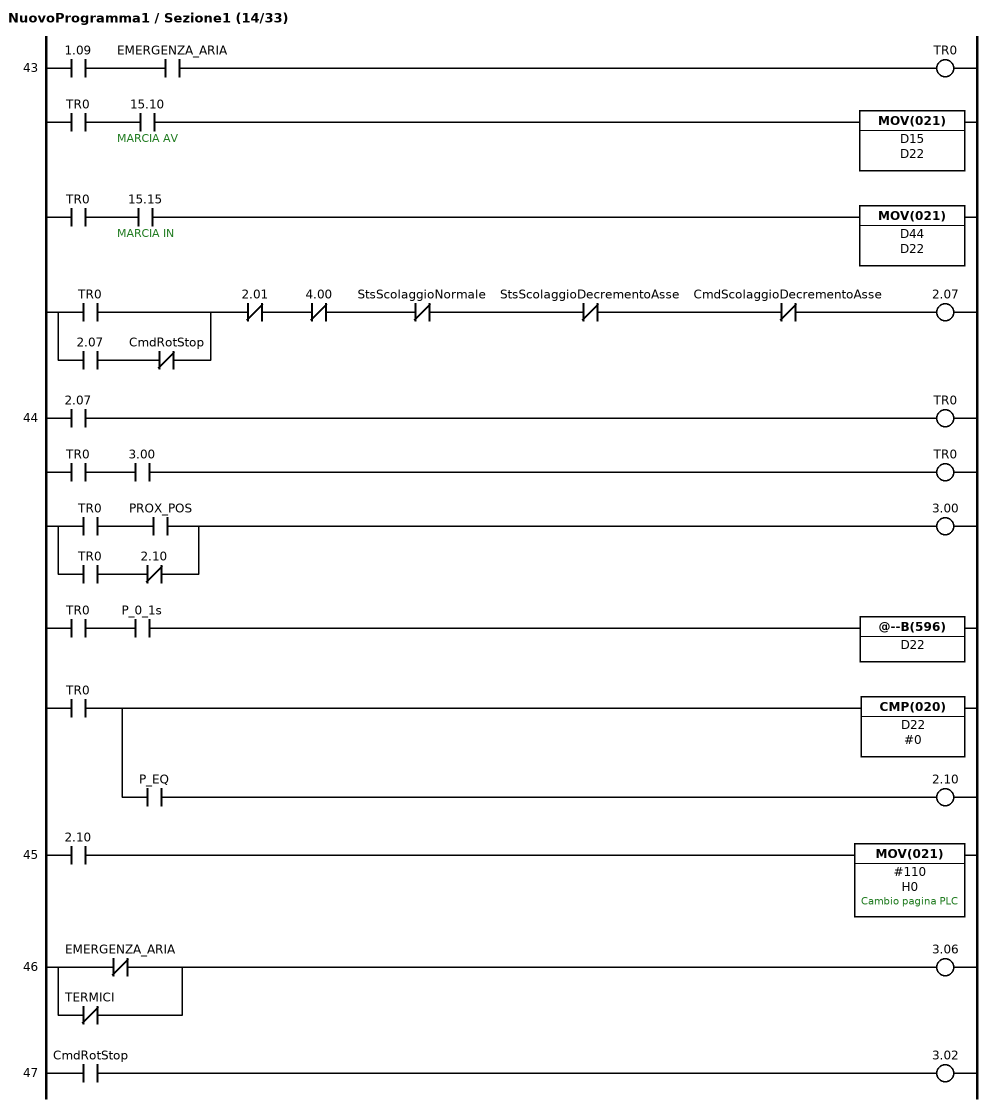
; rung 43
LD 1.09
AND EMERGENZA_ARIA
OUT TR0
AND 15.10  ; MARCIA AV
MOV(021) D15 D22
LD TR0
AND 15.15  ; MARCIA IN
MOV(021) D44 D22
LD TR0
LD 2.07
ANDNOT CmdRotStop
ORLD
ANDNOT 2.01
ANDNOT 4.00
ANDNOT StsScolaggioNormale
ANDNOT StsScolaggioDecrementoAsse
ANDNOT CmdScolaggioDecrementoAsse
OUT 2.07
; rung 44
LD 2.07
OUT TR0
AND PROX_POS
LD TR0
AND 3.00
OUT TR0
ANDNOT 2.10
ORLD
OUT 3.00
LD TR0
AND P_0_1s
@--B(596) D22
LD TR0
CMP(020) D22 #0
AND P_EQ
OUT 2.10
; rung 45
LD 2.10
MOV(021) #110 H0  ; Cambio pagina PLC
; rung 46
LDNOT EMERGENZA_ARIA
ORNOT TERMICI
OUT 3.06
; rung 47
LD CmdRotStop
OUT 3.02

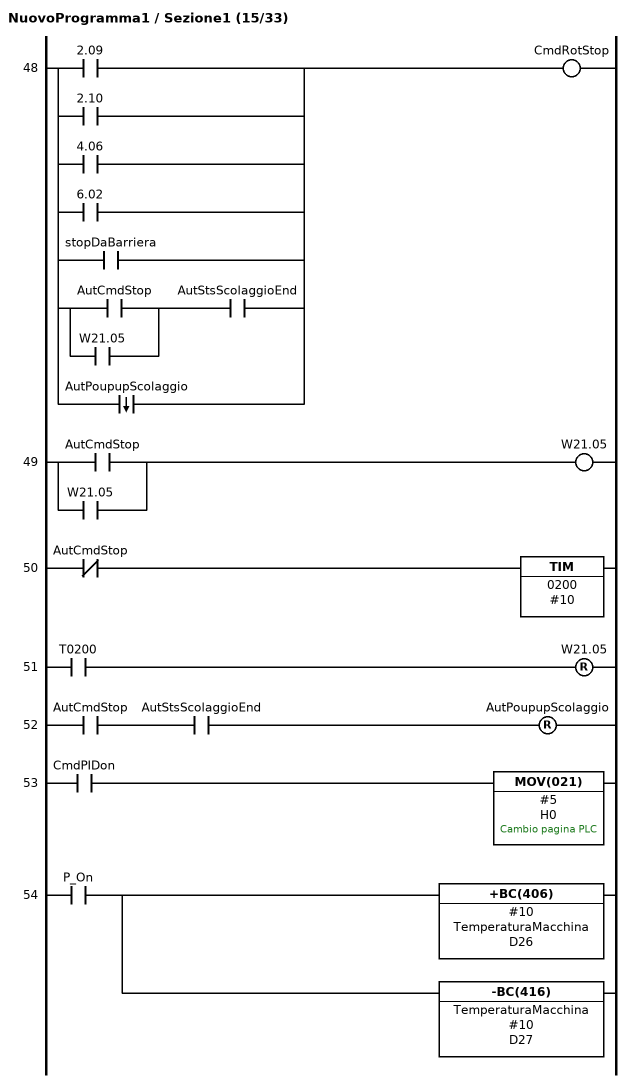
; rung 48
LD 2.09
OR 2.10
OR 4.06
OR 6.02
OR stopDaBarriera
LD AutCmdStop
OR W21.05
AND AutStsScolaggioEnd
ORLD
%OR AutPoupupScolaggio
OUT CmdRotStop
; rung 49
LD AutCmdStop
OR W21.05
OUT W21.05
; rung 50
LDNOT AutCmdStop
TIM 0200 #10
; rung 51
LD T0200
RSET W21.05
; rung 52
LD AutCmdStop
AND AutStsScolaggioEnd
RSET AutPoupupScolaggio
; rung 53
LD CmdPIDon
MOV(021) #5 H0  ; Cambio pagina PLC
; rung 54
LD P_On
+BC(406) #10 TemperaturaMacchina D26
-BC(416) TemperaturaMacchina #10 D27

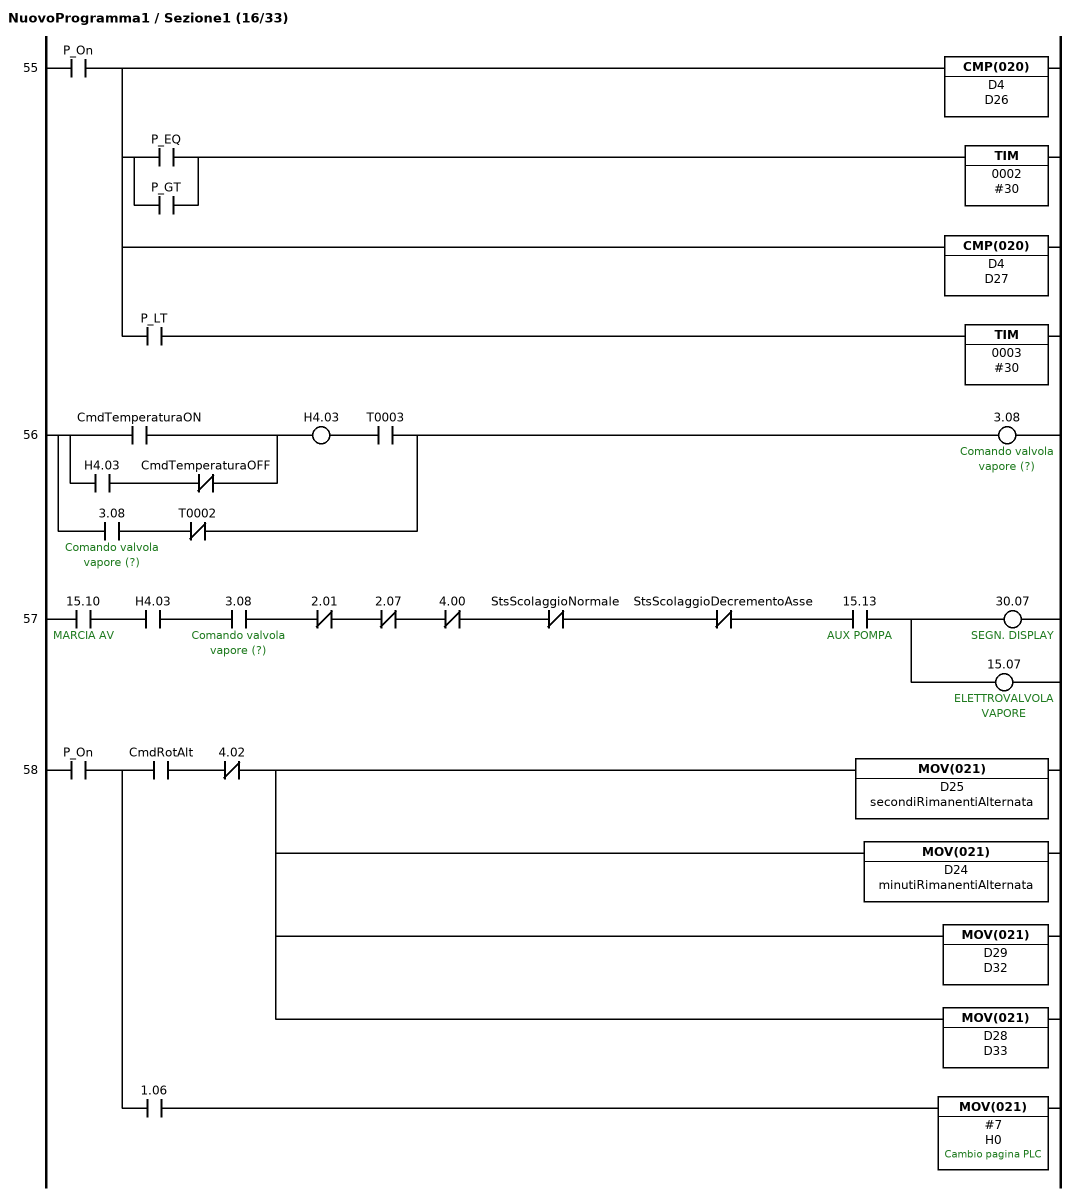
; rung 55
LD P_On
OUT TR0
CMP(020) D4 D26
LD P_EQ
OR P_GT
ANDLD
TIM 0002 #30
LD TR0
CMP(020) D4 D27
AND P_LT
TIM 0003 #30
; rung 56
LD CmdTemperaturaON
LD H4.03
ANDNOT CmdTemperaturaOFF
ORLD
OUT H4.03
AND T0003
LD 3.08  ; Comando valvola vapore (?)
ANDNOT T0002
ORLD
OUT 3.08  ; Comando valvola vapore (?)
; rung 57
LD 15.10  ; MARCIA AV
AND H4.03
AND 3.08  ; Comando valvola vapore (?)
ANDNOT 2.01
ANDNOT 2.07
ANDNOT 4.00
ANDNOT StsScolaggioNormale
ANDNOT StsScolaggioDecrementoAsse
AND 15.13  ; AUX POMPA
OUT 30.07  ; SEGN. DISPLAY
OUT 15.07  ; ELETTROVALVOLA VAPORE
; rung 58
LD P_On
OUT TR0
AND CmdRotAlt
ANDNOT 4.02
MOV(021) D25 secondiRimanentiAlternata
MOV(021) D24 minutiRimanentiAlternata
MOV(021) D29 D32
MOV(021) D28 D33
LD TR0
AND 1.06
MOV(021) #7 H0  ; Cambio pagina PLC

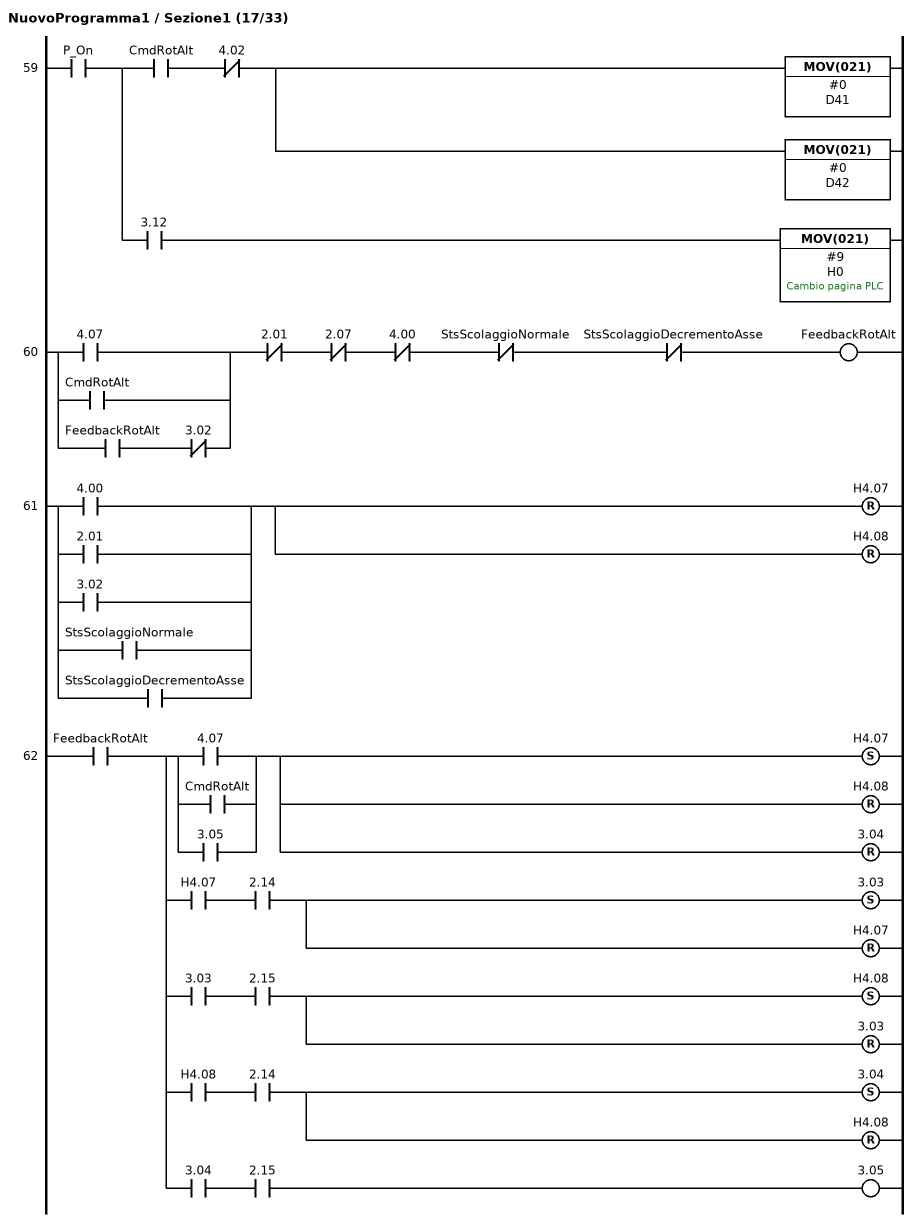
; rung 59
LD P_On
OUT TR0
AND CmdRotAlt
ANDNOT 4.02
MOV(021) #0 D41
MOV(021) #0 D42
LD TR0
AND 3.12
MOV(021) #9 H0  ; Cambio pagina PLC
; rung 60
LD 4.07
OR CmdRotAlt
LD FeedbackRotAlt
ANDNOT 3.02
ORLD
ANDNOT 2.01
ANDNOT 2.07
ANDNOT 4.00
ANDNOT StsScolaggioNormale
ANDNOT StsScolaggioDecrementoAsse
OUT FeedbackRotAlt
; rung 61
LD 4.00
OR 2.01
OR 3.02
OR StsScolaggioNormale
OR StsScolaggioDecrementoAsse
RSET H4.07
RSET H4.08
; rung 62
LD FeedbackRotAlt
OUT TR0
LD 4.07
OR CmdRotAlt
OR 3.05
ANDLD
SET H4.07
RSET H4.08
RSET 3.04
LD TR0
AND H4.07
AND 2.14
SET 3.03
RSET H4.07
LD TR0
AND 3.03
AND 2.15
SET H4.08
RSET 3.03
LD TR0
AND H4.08
AND 2.14
SET 3.04
RSET H4.08
LD TR0
AND 3.04
AND 2.15
OUT 3.05

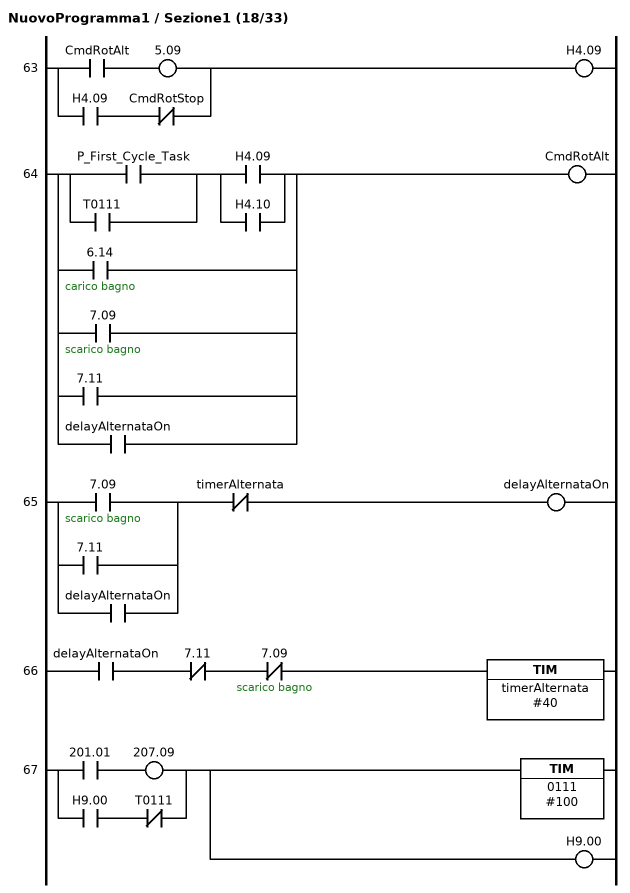
; rung 63
LD CmdRotAlt
OUT 5.09
LD H4.09
ANDNOT CmdRotStop
ORLD
OUT H4.09
; rung 64
LD P_First_Cycle_Task
OR T0111
LD H4.09
OR H4.10
ANDLD
OR 6.14  ; carico bagno
OR 7.09  ; scarico bagno
OR 7.11
OR delayAlternataOn
OUT CmdRotAlt
; rung 65
LD 7.09  ; scarico bagno
OR 7.11
OR delayAlternataOn
ANDNOT timerAlternata
OUT delayAlternataOn
; rung 66
LD delayAlternataOn
ANDNOT 7.11
ANDNOT 7.09  ; scarico bagno
TIM timerAlternata #40
; rung 67
LD 201.01
OUT 207.09
LD H9.00
ANDNOT T0111
ORLD
TIM 0111 #100
OUT H9.00

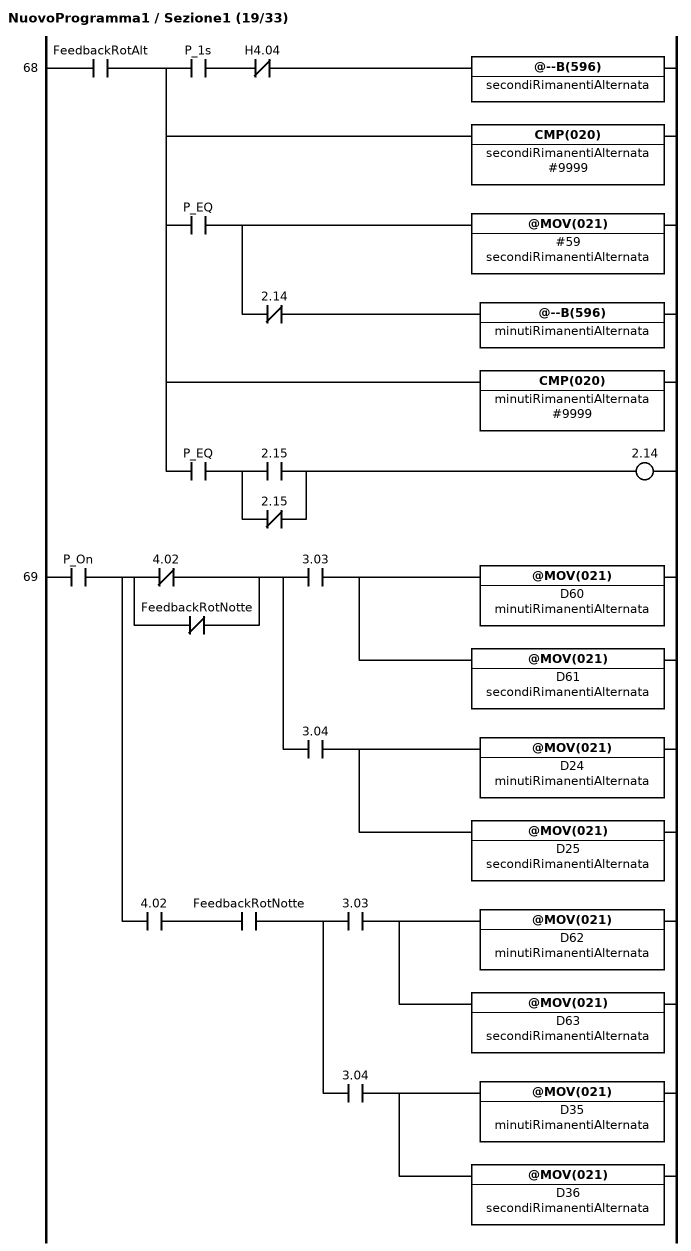
; rung 68
LD FeedbackRotAlt
OUT TR0
AND P_1s
ANDNOT H4.04
@--B(596) secondiRimanentiAlternata
LD TR0
CMP(020) secondiRimanentiAlternata #9999
AND P_EQ
@MOV(021) #59 secondiRimanentiAlternata
ANDNOT 2.14
@--B(596) minutiRimanentiAlternata
LD TR0
CMP(020) minutiRimanentiAlternata #9999
AND P_EQ
LD 2.15
ORNOT 2.15
ANDLD
OUT 2.14
; rung 69
LD P_On
OUT TR0
LDNOT 4.02
ORNOT FeedbackRotNotte
ANDLD
OUT TR1
AND 3.03
@MOV(021) D60 minutiRimanentiAlternata
@MOV(021) D61 secondiRimanentiAlternata
LD TR1
AND 3.04
@MOV(021) D24 minutiRimanentiAlternata
@MOV(021) D25 secondiRimanentiAlternata
LD TR0
AND 4.02
AND FeedbackRotNotte
OUT TR0
AND 3.03
@MOV(021) D62 minutiRimanentiAlternata
@MOV(021) D63 secondiRimanentiAlternata
LD TR0
AND 3.04
@MOV(021) D35 minutiRimanentiAlternata
@MOV(021) D36 secondiRimanentiAlternata

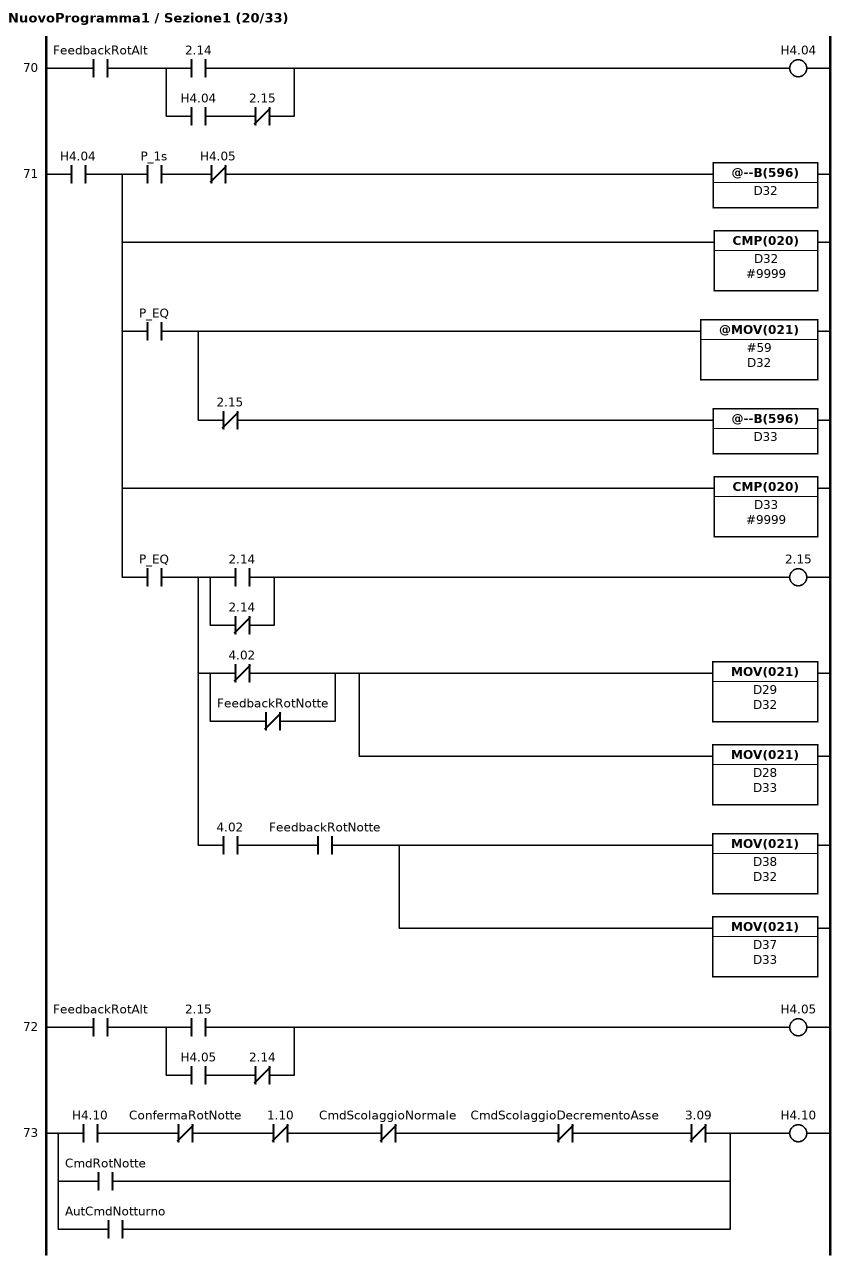
; rung 70
LD FeedbackRotAlt
LD 2.14
LD H4.04
ANDNOT 2.15
ORLD
ANDLD
OUT H4.04
; rung 71
LD H4.04
OUT TR0
AND P_1s
ANDNOT H4.05
@--B(596) D32
LD TR0
CMP(020) D32 #9999
AND P_EQ
@MOV(021) #59 D32
ANDNOT 2.15
@--B(596) D33
LD TR0
CMP(020) D33 #9999
AND P_EQ
OUT TR0
LD 2.14
ORNOT 2.14
ANDLD
OUT 2.15
LD TR0
LDNOT 4.02
ORNOT FeedbackRotNotte
ANDLD
MOV(021) D29 D32
MOV(021) D28 D33
LD TR0
AND 4.02
AND FeedbackRotNotte
MOV(021) D38 D32
MOV(021) D37 D33
; rung 72
LD FeedbackRotAlt
LD 2.15
LD H4.05
ANDNOT 2.14
ORLD
ANDLD
OUT H4.05
; rung 73
LD H4.10
ANDNOT ConfermaRotNotte
ANDNOT 1.10
ANDNOT CmdScolaggioNormale
ANDNOT CmdScolaggioDecrementoAsse
ANDNOT 3.09
OR CmdRotNotte
OR AutCmdNotturno
OUT H4.10

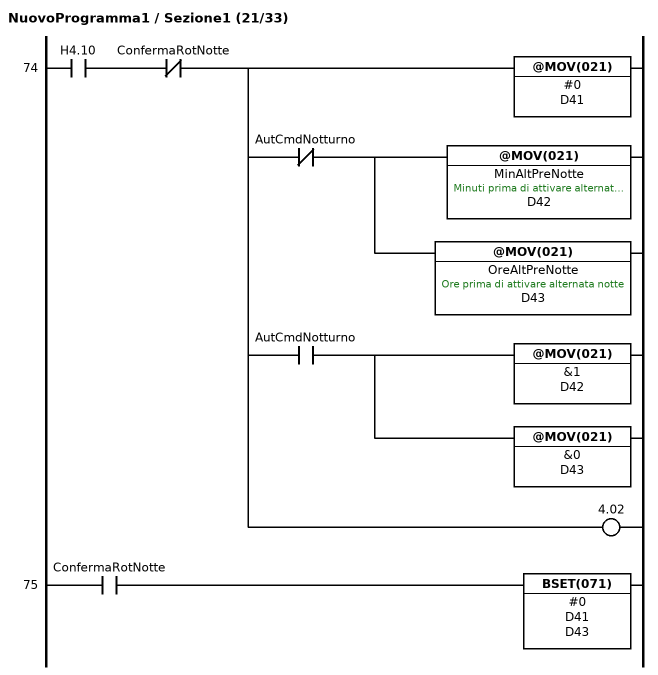
; rung 74
LD H4.10
ANDNOT ConfermaRotNotte
OUT TR0
@MOV(021) #0 D41
ANDNOT AutCmdNotturno
@MOV(021) MinAltPreNotte D42  ; Minuti prima di attivare alternata notte
@MOV(021) OreAltPreNotte D43  ; Ore prima di attivare alternata notte
LD TR0
AND AutCmdNotturno
@MOV(021) &1 D42
@MOV(021) &0 D43
LD TR0
OUT 4.02
; rung 75
LD ConfermaRotNotte
BSET(071) #0 D41 D43

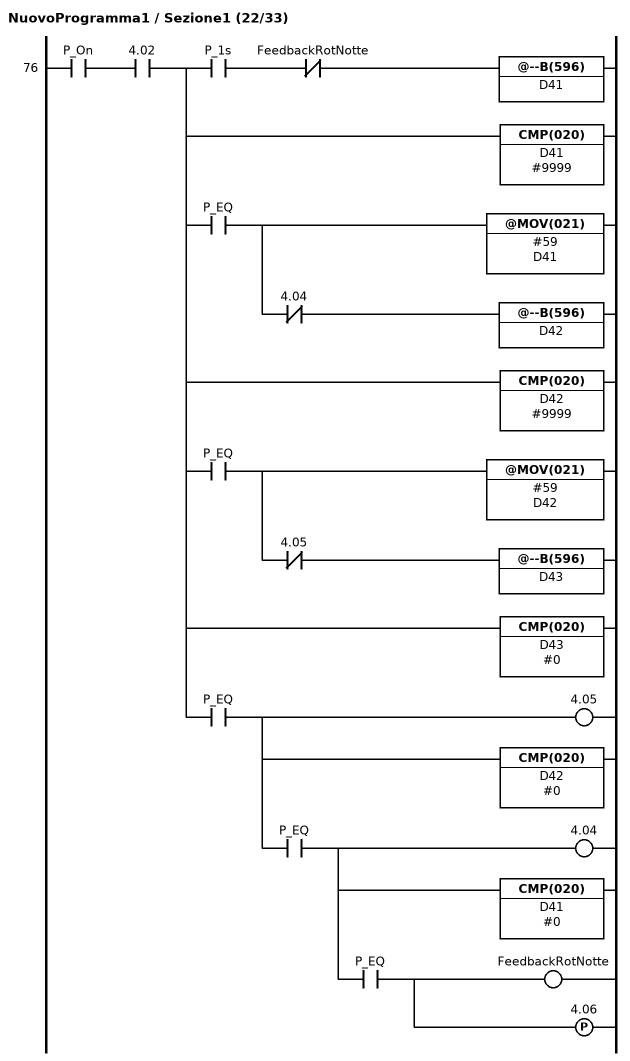
; rung 76
LD P_On
AND 4.02
OUT TR0
AND P_1s
ANDNOT FeedbackRotNotte
@--B(596) D41
LD TR0
CMP(020) D41 #9999
AND P_EQ
@MOV(021) #59 D41
ANDNOT 4.04
@--B(596) D42
LD TR0
CMP(020) D42 #9999
AND P_EQ
@MOV(021) #59 D42
ANDNOT 4.05
@--B(596) D43
LD TR0
CMP(020) D43 #0
AND P_EQ
OUT 4.05
CMP(020) D42 #0
AND P_EQ
OUT 4.04
CMP(020) D41 #0
AND P_EQ
OUT FeedbackRotNotte
DIFU(013) 4.06

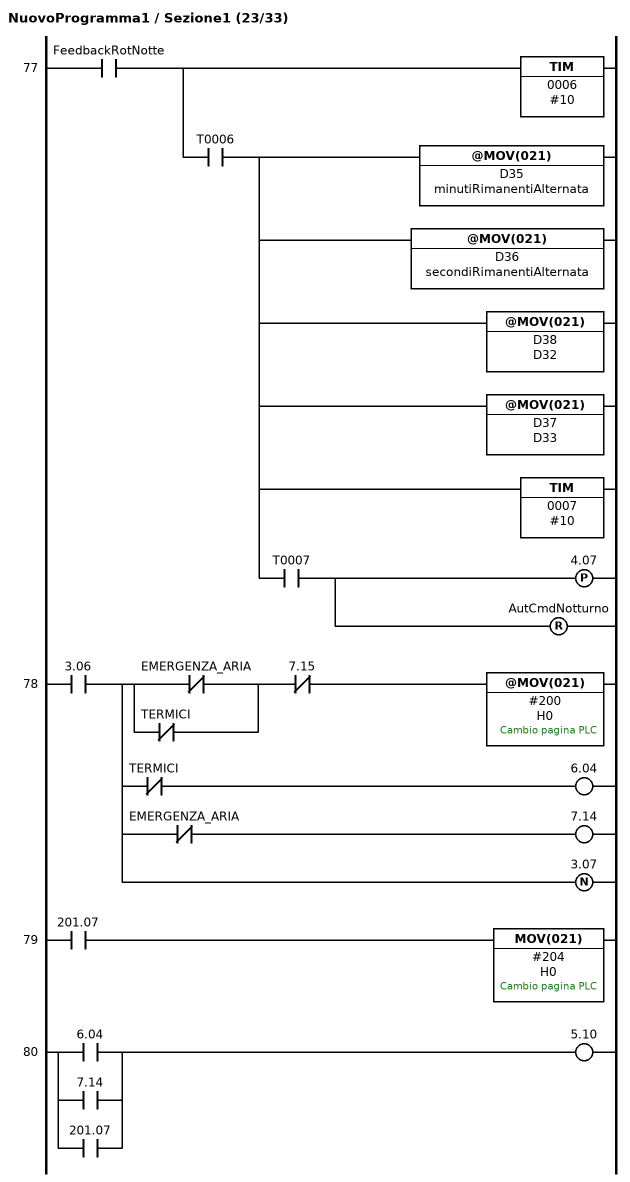
; rung 77
LD FeedbackRotNotte
TIM 0006 #10
AND T0006
@MOV(021) D35 minutiRimanentiAlternata
@MOV(021) D36 secondiRimanentiAlternata
@MOV(021) D38 D32
@MOV(021) D37 D33
TIM 0007 #10
AND T0007
DIFU(013) 4.07
RSET AutCmdNotturno
; rung 78
LD 3.06
OUT TR0
LDNOT EMERGENZA_ARIA
ORNOT TERMICI
ANDLD
ANDNOT 7.15
@MOV(021) #200 H0  ; Cambio pagina PLC
LD TR0
ANDNOT TERMICI
OUT 6.04
LD TR0
ANDNOT EMERGENZA_ARIA
OUT 7.14
LD TR0
DIFD(014) 3.07
; rung 79
LD 201.07
MOV(021) #204 H0  ; Cambio pagina PLC
; rung 80
LD 6.04
OR 7.14
OR 201.07
OUT 5.10

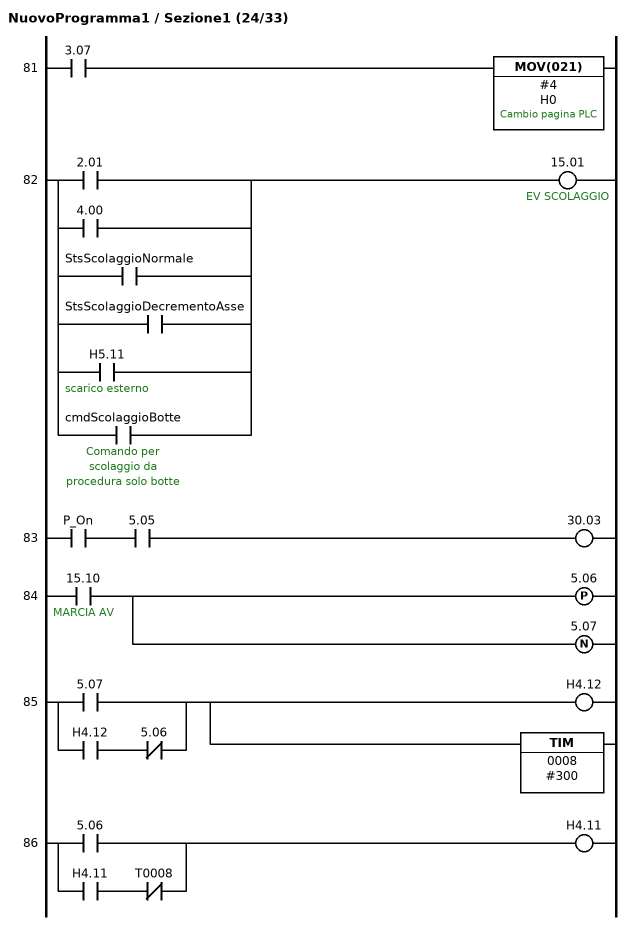
; rung 81
LD 3.07
MOV(021) #4 H0  ; Cambio pagina PLC
; rung 82
LD 2.01
OR 4.00
OR StsScolaggioNormale
OR StsScolaggioDecrementoAsse
OR H5.11  ; scarico esterno
OR cmdScolaggioBotte  ; Comando per scolaggio da procedura solo botte
OUT 15.01  ; EV SCOLAGGIO
; rung 83
LD P_On
AND 5.05
OUT 30.03
; rung 84
LD 15.10  ; MARCIA AV
DIFU(013) 5.06
DIFD(014) 5.07
; rung 85
LD 5.07
LD H4.12
ANDNOT 5.06
ORLD
OUT H4.12
TIM 0008 #300
; rung 86
LD 5.06
LD H4.11
ANDNOT T0008
ORLD
OUT H4.11

